TYPE DUT_SENSOR_DATAS_h4 :
UNION
	data_lreal:REAL;
	data_byte:ARRAY[0..3] OF BYTE;
END_UNION
END_TYPE

(* stored: Version 1.1.0.1, ProductVersion 3.1.4024.6
   DUT DUT_SENSOR_DATAS_h4: Id {7f0cb130-0a1c-4c2b-b126-d8b8d2a9d86c} *)
